// TIA Portal project "PLCII_Pro7" (V15.1)

(* hardware
DEVICE "S7-1200 station_1"  S7-1200 Station
   slot 0: "Rack_0"  S7-1200 Rack  Rack  V1.0
   slot 1: "PLC_1"  CPU 1215C DC/DC/Rly  6ES7 215-1HG40-0XB0  V4.2
*)

// ===== PLC "PLC_1"  CPU 1215C DC/DC/Rly =====

VAR_GLOBAL   // PLC tag table "Default tag table"
   "Start" AT %M0.0 : Bool;
   "Sys_runing" AT %M0.1 : Bool;
   "Stop" AT %M0.2 : Bool;
   "Activate" AT %M0.3 : Bool;
   "Sys_Activated" AT %M0.4 : Bool;
END_VAR

DATA_BLOCK "SysVaribales"   // DB1
{ S7_Optimized_Access := 'TRUE' }
VERSION : 0.1
   VAR
      StartSampling : Bool;
      StopSampling : Bool;
      SamplingRuning : Bool;
      StartCalibraton : Bool;
      StopCalibration : Bool;
      CalibrationRuning : Bool;
      O2Concentration : Int;
      O2ConcentrationMesuered : Int;
      O2_30Valve : Bool;
      O2_00Valve : Bool;
      StartCalibrationSeq : Bool;
      CalibrationDone : Bool;
      ScaleInputMIN : Int;
      ScaleInputMAX : Int := 0;
      O2_Zero_Average : Int;
      "O2_Maximum_ Concentration" : Int;
      "O2_Calibration_Gas_ Concentration" : Int;
      O2_Test_Gas_Average : Int;
      O2_Mesured : Int;
      O2_Concentration : Int;
   END_VAR
BEGIN
END_DATA_BLOCK

DATA_BLOCK "Sampling&&Calibration_DB"   // DB2
{ S7_Optimized_Access := 'TRUE' }
VERSION : 0.1
// stored: InstanceOfName Sampling&&Calibration
"Sampling&&Calibration"
BEGIN
END_DATA_BLOCK

DATA_BLOCK "ActuateValves_DB"   // DB5
{ S7_Optimized_Access := 'TRUE' }
VERSION : 0.1
// stored: InstanceOfName Calibration
"Calibration"
BEGIN
END_DATA_BLOCK

DATA_BLOCK "Calibration_DB"   // DB6
{ S7_Optimized_Access := 'TRUE' }
VERSION : 0.1
// stored: InstanceOfName Calibration
"Calibration"
BEGIN
END_DATA_BLOCK

DATA_BLOCK "Sampling_DB"   // DB7
{ S7_Optimized_Access := 'TRUE' }
VERSION : 0.1
// stored: InstanceOfName Sampling
"Sampling"
BEGIN
END_DATA_BLOCK

// folder: System blocks/Program resources

DATA_BLOCK "IEC_Timer_0_DB"   // DB3
{ S7_Optimized_Access := 'TRUE' }
AUTHOR : Simatic
FAMILY : IEC
NAME : IEC_TMR
VERSION : 1.0
// stored: InstanceOfName IEC_TIMER
"IEC_TIMER"
BEGIN
END_DATA_BLOCK

DATA_BLOCK "IEC_Timer_0_DB_1"   // DB4
{ S7_Optimized_Access := 'TRUE' }
AUTHOR : Simatic
FAMILY : IEC
NAME : IEC_TMR
VERSION : 1.0
// stored: InstanceOfName IEC_TIMER
"IEC_TIMER"
BEGIN
END_DATA_BLOCK

// folder: (top level)

FUNCTION_BLOCK "Sampling&&Calibration"   // FB1, LAD
{ S7_Optimized_Access := 'TRUE' }
VERSION : 0.1
   VAR_INPUT
      O2_Measured : Int;
   END_VAR
   VAR_OUTPUT
      O2_Concenetration : Real;
   END_VAR
   VAR
      ons1 : Bool;
      ons2 : Bool;
      ons3 : Bool;
      ons4 : Bool;
      ons5 : Bool;
      ons6 : Bool;
      ons7 : Bool;
      ons8 : Bool;
      ons9 : Bool;
      ons10 : Bool;
      ons11 : Bool;
   END_VAR
   VAR_TEMP
      O2_ValueTreated : Real;
   END_VAR
   VAR_TEMP   // added for the SCL form of the ladder/FBD networks
      _w1 : Bool;
   END_VAR
BEGIN

REGION Network 1
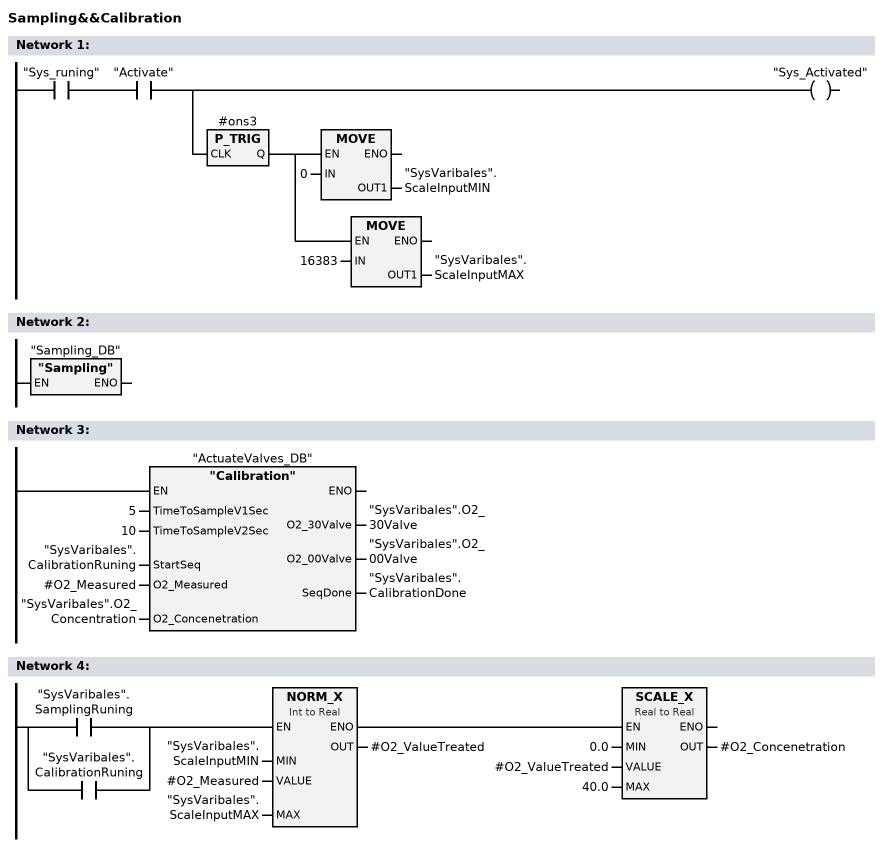
   RUNG wire#powerrail
      Contact( "Sys_runing" )
      Contact( "Activate" )
      wire#w1
      Coil( "Sys_Activated" )
   END_RUNG
   RUNG wire#w1
      P_Trig( #ons3 )
      wire#w2
      Move(in := 0, out1 => "SysVaribales".ScaleInputMIN)
   END_RUNG
   RUNG wire#w2
      Move(in := 16383, out1 => "SysVaribales".ScaleInputMAX)
   END_RUNG
   // the same network as SCL:
   "Sys_Activated" := "Sys_runing" AND "Activate";
   #_w1 := "Sys_Activated" AND NOT #ons3;   // rising edge
   #ons3 := "Sys_Activated";
   IF #_w1 THEN
       "SysVaribales".ScaleInputMIN := 0;
       "SysVaribales".ScaleInputMAX := 16383;
   END_IF;
END_REGION

REGION Network 2
   RUNG wire#powerrail
      "Sampling_DB"()
   END_RUNG
   // the same network as SCL:
   "Sampling_DB"();   // "Sampling"
END_REGION

REGION Network 3
   RUNG wire#powerrail
      "ActuateValves_DB"(TimeToSampleV1Sec := 5, TimeToSampleV2Sec := 10, StartSeq := "SysVaribales".CalibrationRuning, O2_Measured := #O2_Measured, O2_Concenetration := "SysVaribales".O2_Concentration, O2_30Valve => "SysVaribales".O2_30Valve, O2_00Valve => "SysVaribales".O2_00Valve, SeqDone => "SysVaribales".CalibrationDone)
   END_RUNG
   // the same network as SCL:
   "ActuateValves_DB"(TimeToSampleV1Sec := 5,   // "Calibration"
                      TimeToSampleV2Sec := 10,
                      StartSeq := "SysVaribales".CalibrationRuning,
                      O2_Measured := #O2_Measured,
                      O2_Concenetration := "SysVaribales".O2_Concentration,
                      O2_30Valve => "SysVaribales".O2_30Valve,
                      O2_00Valve => "SysVaribales".O2_00Valve,
                      SeqDone => "SysVaribales".CalibrationDone);
END_REGION

REGION Network 4
   RUNG wire#powerrail
      Contact( "SysVaribales".SamplingRuning )
      wire#w1
      { S7_Templates := "[SrcType := Int, DestType := Real]" } Normalize(min := "SysVaribales".ScaleInputMIN, value := #O2_Measured, max := "SysVaribales".ScaleInputMAX, out => #O2_ValueTreated)
      { S7_Templates := "[SrcType := Real, DestType := Real]" } Scale(min := 0.0, value := #O2_ValueTreated, max := 40.0, out => #O2_Concenetration)
   END_RUNG
   RUNG wire#powerrail
      Contact( "SysVaribales".CalibrationRuning )
   END_RUNG wire#w1
   // the same network as SCL:
   IF "SysVaribales".SamplingRuning OR "SysVaribales".CalibrationRuning THEN
       #O2_ValueTreated := NORM_X(MIN := "SysVaribales".ScaleInputMIN, VALUE := #O2_Measured, MAX := "SysVaribales".ScaleInputMAX);
       #O2_Concenetration := SCALE_X(MIN := 0.0, VALUE := #O2_ValueTreated, MAX := 40.0);
   END_IF;
END_REGION
END_FUNCTION_BLOCK

FUNCTION_BLOCK "Calibration"   // FB2, LAD
{ S7_Optimized_Access := 'TRUE' }
VERSION : 0.1
   VAR_INPUT
      TimeToSampleV1Sec : Int;
      TimeToSampleV2Sec : Int;
      StartSeq : Bool;
      O2_Measured : Int;
   END_VAR
   VAR_OUTPUT
      O2_30Valve : Bool;
      O2_00Valve : Bool;
      SeqDone : Bool;
   END_VAR
   VAR_IN_OUT
      O2_Concenetration : Int;
   END_VAR
   VAR
      startSecValve : Bool;
      ons1 : Bool;
      ons2 : Bool;
      ons3 : Bool;
      ons4 : Bool;
      ons5 : Bool;
      ons6 : Bool;
      ons7 : Bool;
      ons8 : Bool;
      UsedTIme1 : Time;
      UsedTIme2 : Time;
      O2_ValueTreated2 : Real;
   END_VAR
   VAR_TEMP
      TimeTemp1 : Int;
      UsedTimeTemp1 : Time;
      TimeTemp2 : Int;
      UsedTimeTemp2 : Time;
      O2_ValueTreated : Real;
      O2_30Average_MaxScaleTemp : Int;
      "O2_Maximum_ ConcentrationTemp" : Int;
      ScaleInputMAXTemp : Int;
      ScaleInputMAXTempReal : Real;
      ScaleInputMAXTempINT : Int;
   END_VAR
   VAR_TEMP   // added for the SCL form of the ladder/FBD networks
      _w1 : Bool;
      _w2 : Bool;
   END_VAR
BEGIN

REGION Network 1
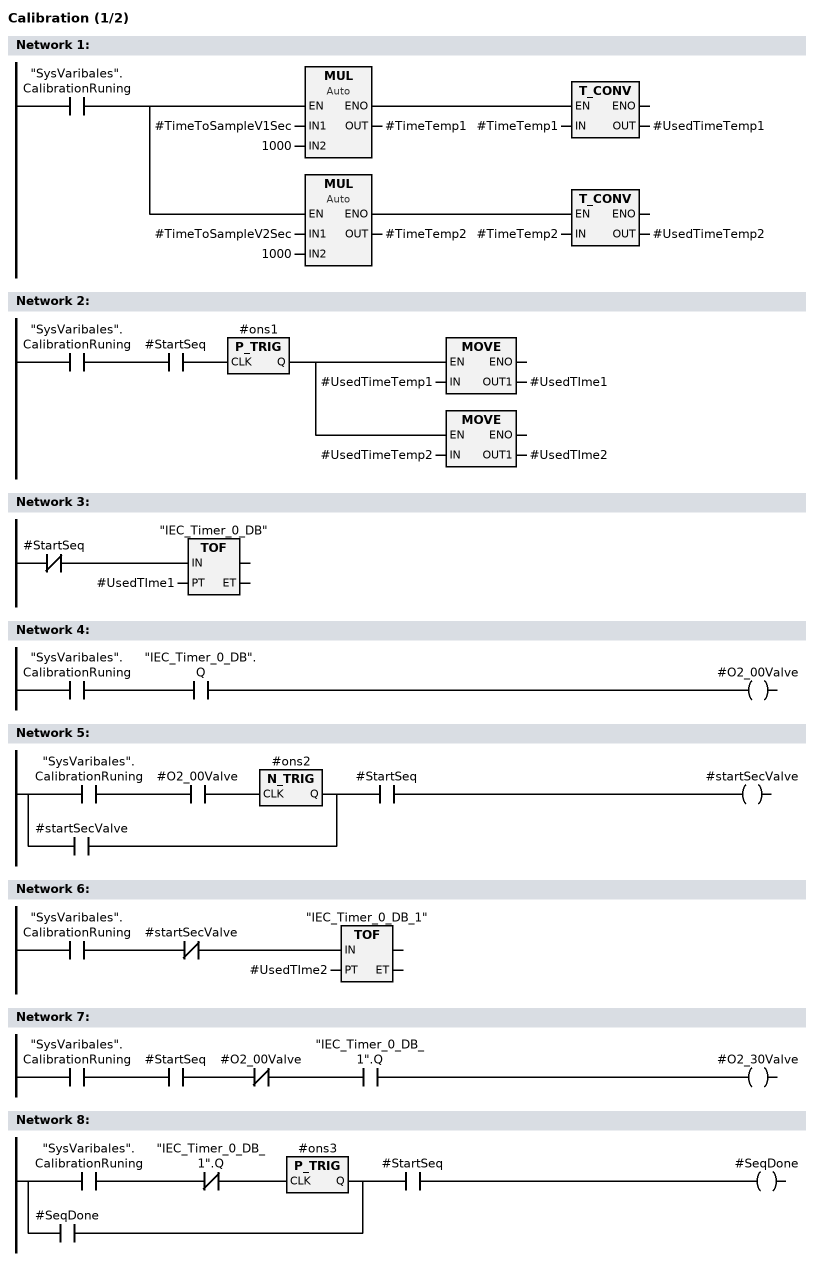
   IF "SysVaribales".CalibrationRuning THEN #TimeTemp1 := #TimeToSampleV1Sec * 1000; END_IF;
   #_w1 := "SysVaribales".CalibrationRuning;
   IF #_w1 THEN
       #UsedTimeTemp1 := T_CONV(IN := #TimeTemp1);
       #TimeTemp2 := #TimeToSampleV2Sec * 1000;
       #UsedTimeTemp2 := T_CONV(IN := #TimeTemp2);
   END_IF;
END_REGION

REGION Network 2
   RUNG wire#powerrail
      Contact( "SysVaribales".CalibrationRuning )
      Contact( #StartSeq )
      P_Trig( #ons1 )
      wire#w1
      Move(in := #UsedTimeTemp1, out1 => #UsedTIme1)
   END_RUNG
   RUNG wire#w1
      Move(in := #UsedTimeTemp2, out1 => #UsedTIme2)
   END_RUNG
   // the same network as SCL:
   #_w1 := "SysVaribales".CalibrationRuning AND #StartSeq;
   #_w2 := #_w1 AND NOT #ons1;   // rising edge
   #ons1 := #_w1;
   IF #_w2 THEN
       #UsedTIme1 := #UsedTimeTemp1;
       #UsedTIme2 := #UsedTimeTemp2;
   END_IF;
END_REGION

REGION Network 3
   "IEC_Timer_0_DB".TOF(IN := NOT #StartSeq, PT := #UsedTIme1);
END_REGION

REGION Network 4
   RUNG wire#powerrail
      Contact( "SysVaribales".CalibrationRuning )
      Contact( "IEC_Timer_0_DB".Q )
      Coil( #O2_00Valve )
   END_RUNG
   // the same network as SCL:
   #O2_00Valve := "SysVaribales".CalibrationRuning AND "IEC_Timer_0_DB".Q;
END_REGION

REGION Network 5
   RUNG wire#powerrail
      Contact( "SysVaribales".CalibrationRuning )
      Contact( #O2_00Valve )
      N_Trig( #ons2 )
      wire#w1
      Contact( #StartSeq )
      Coil( #startSecValve )
   END_RUNG
   RUNG wire#powerrail
      Contact( #startSecValve )
   END_RUNG wire#w1
   // the same network as SCL:
   #_w1 := "SysVaribales".CalibrationRuning AND #O2_00Valve;
   #_w2 := NOT #_w1 AND #ons2;   // falling edge
   #ons2 := #_w1;
   #startSecValve := (#_w2 OR #startSecValve) AND #StartSeq;
END_REGION

REGION Network 6
   "IEC_Timer_0_DB_1".TOF(IN := "SysVaribales".CalibrationRuning AND NOT #startSecValve, PT := #UsedTIme2);
END_REGION

REGION Network 7
   RUNG wire#powerrail
      Contact( "SysVaribales".CalibrationRuning )
      Contact( #StartSeq )
      I_Contact( #O2_00Valve )
      Contact( "IEC_Timer_0_DB_1".Q )
      Coil( #O2_30Valve )
   END_RUNG
   // the same network as SCL:
   #O2_30Valve := "SysVaribales".CalibrationRuning AND #StartSeq AND NOT #O2_00Valve AND "IEC_Timer_0_DB_1".Q;
END_REGION

REGION Network 8
   RUNG wire#powerrail
      Contact( "SysVaribales".CalibrationRuning )
      I_Contact( "IEC_Timer_0_DB_1".Q )
      P_Trig( #ons3 )
      wire#w1
      Contact( #StartSeq )
      Coil( #SeqDone )
   END_RUNG
   RUNG wire#powerrail
      Contact( #SeqDone )
   END_RUNG wire#w1
   // the same network as SCL:
   #_w1 := "SysVaribales".CalibrationRuning AND NOT "IEC_Timer_0_DB_1".Q;
   #_w2 := #_w1 AND NOT #ons3;   // rising edge
   #ons3 := #_w1;
   #SeqDone := (#_w2 OR #SeqDone) AND #StartSeq;
END_REGION

REGION Network 9
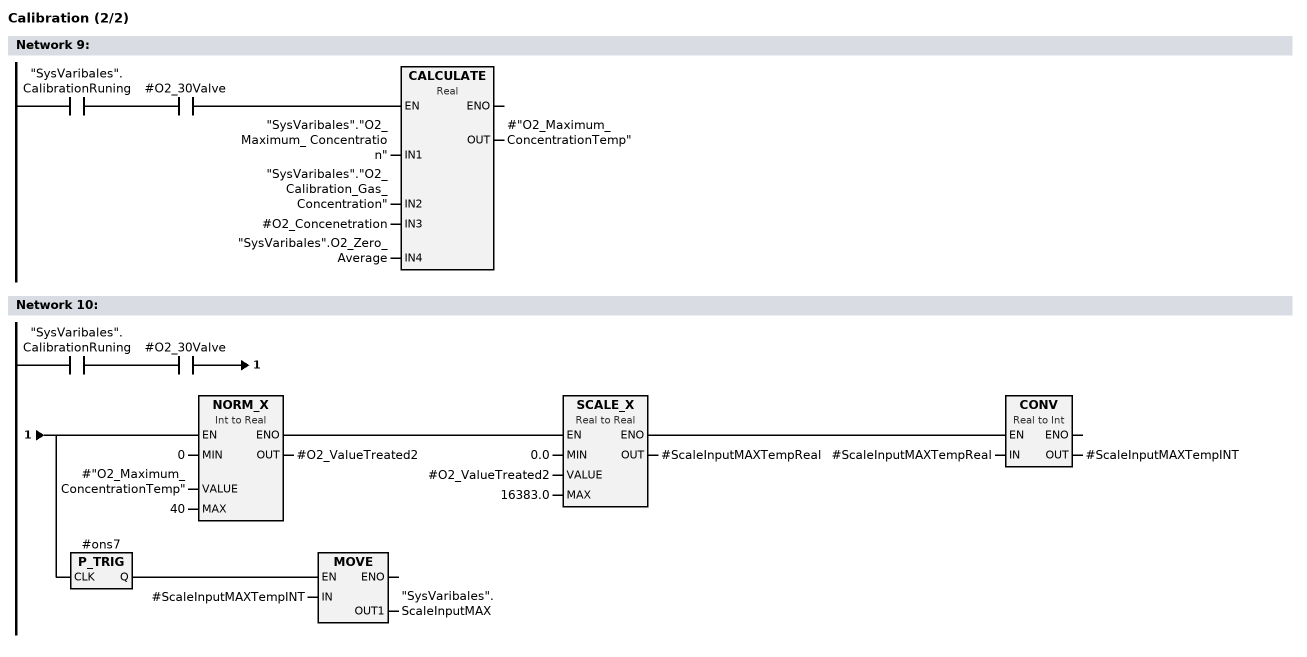
   RUNG wire#powerrail
      Contact( "SysVaribales".CalibrationRuning )
      Contact( #O2_30Valve )
      { S7_Templates := "SrcType := Real"; S7_Expression := "((IN1/IN2)*(IN3-IN4)) + IN4" } Calculate(in1 := "SysVaribales"."O2_Maximum_ Concentration", in2 := "SysVaribales"."O2_Calibration_Gas_ Concentration", in3 := #O2_Concenetration, in4 := "SysVaribales".O2_Zero_Average, out => #"O2_Maximum_ ConcentrationTemp")
   END_RUNG
   // the same network as SCL:
   IF "SysVaribales".CalibrationRuning AND #O2_30Valve THEN
       #"O2_Maximum_ ConcentrationTemp" := (("SysVaribales"."O2_Maximum_ Concentration"/"SysVaribales"."O2_Calibration_Gas_ Concentration")*(#O2_Concenetration-"SysVaribales".O2_Zero_Average)) + "SysVaribales".O2_Zero_Average;
   END_IF;
END_REGION

REGION Network 10
   RUNG wire#powerrail
      Contact( "SysVaribales".CalibrationRuning )
      Contact( #O2_30Valve )
      wire#w1
      { S7_Templates := "[SrcType := Int, DestType := Real]" } Normalize(min := 0, value := #"O2_Maximum_ ConcentrationTemp", max := 40, out => #O2_ValueTreated2)
      { S7_Templates := "[SrcType := Real, DestType := Real]" } Scale(min := 0.0, value := #O2_ValueTreated2, max := 16383.0, out => #ScaleInputMAXTempReal)
      { S7_Templates := "[SrcType := Real, DestType := Int]" } Convert(in := #ScaleInputMAXTempReal, out => #ScaleInputMAXTempINT)
   END_RUNG
   RUNG wire#w1
      P_Trig( #ons7 )
      Move(in := #ScaleInputMAXTempINT, out1 => "SysVaribales".ScaleInputMAX)
   END_RUNG
   // the same network as SCL:
   #_w1 := "SysVaribales".CalibrationRuning AND #O2_30Valve;
   IF #_w1 THEN
       #O2_ValueTreated2 := NORM_X(MIN := 0, VALUE := #"O2_Maximum_ ConcentrationTemp", MAX := 40);
       #ScaleInputMAXTempReal := SCALE_X(MIN := 0.0, VALUE := #O2_ValueTreated2, MAX := 16383.0);
       #ScaleInputMAXTempINT := REAL_TO_INT(#ScaleInputMAXTempReal);
   END_IF;
   #_w2 := #_w1 AND NOT #ons7;   // rising edge
   #ons7 := #_w1;
   IF #_w2 THEN "SysVaribales".ScaleInputMAX := #ScaleInputMAXTempINT; END_IF;
END_REGION
END_FUNCTION_BLOCK

FUNCTION_BLOCK "Sampling"   // FB3, LAD
{ S7_Optimized_Access := 'TRUE' }
VERSION : 0.1
   VAR
      ons1 : Bool;
      ons2 : Bool;
      ons3 : Bool;
      ons4 : Bool;
      ons5 : Bool;
      ons6 : Bool;
      ons7 : Bool;
      ons8 : Bool;
   END_VAR
   VAR_TEMP   // added for the SCL form of the ladder/FBD networks
      _w1 : Bool;
   END_VAR
BEGIN

REGION Network 1
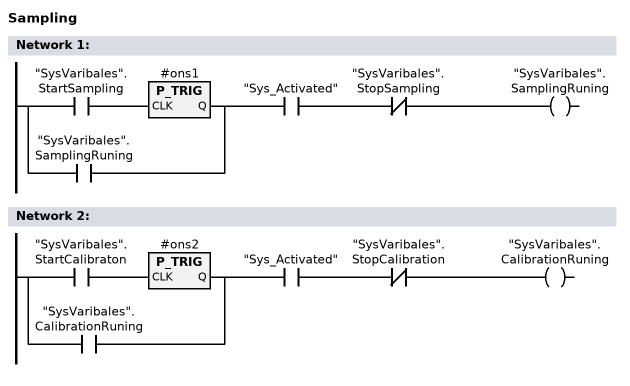
   RUNG wire#powerrail
      Contact( "SysVaribales".StartSampling )
      P_Trig( #ons1 )
      wire#w1
      Contact( "Sys_Activated" )
      I_Contact( "SysVaribales".StopSampling )
      Coil( "SysVaribales".SamplingRuning )
   END_RUNG
   RUNG wire#powerrail
      Contact( "SysVaribales".SamplingRuning )
   END_RUNG wire#w1
   // the same network as SCL:
   #_w1 := "SysVaribales".StartSampling AND NOT #ons1;   // rising edge
   #ons1 := "SysVaribales".StartSampling;
   "SysVaribales".SamplingRuning := (#_w1 OR "SysVaribales".SamplingRuning) AND "Sys_Activated" AND NOT "SysVaribales".StopSampling;
END_REGION

REGION Network 2
   RUNG wire#powerrail
      Contact( "SysVaribales".StartCalibraton )
      P_Trig( #ons2 )
      wire#w1
      Contact( "Sys_Activated" )
      I_Contact( "SysVaribales".StopCalibration )
      Coil( "SysVaribales".CalibrationRuning )
   END_RUNG
   RUNG wire#powerrail
      Contact( "SysVaribales".CalibrationRuning )
   END_RUNG wire#w1
   // the same network as SCL:
   #_w1 := "SysVaribales".StartCalibraton AND NOT #ons2;   // rising edge
   #ons2 := "SysVaribales".StartCalibraton;
   "SysVaribales".CalibrationRuning := (#_w1 OR "SysVaribales".CalibrationRuning) AND "Sys_Activated" AND NOT "SysVaribales".StopCalibration;
END_REGION
END_FUNCTION_BLOCK

ORGANIZATION_BLOCK "Main"   // OB1, LAD, ProgramCycle
TITLE = "Main Program Sweep (Cycle)"
{ S7_Optimized_Access := 'TRUE' }
VERSION : 0.1
   VAR_INPUT
      Initial_Call : Bool;   // Initial call of this OB
      Remanence : Bool;   // =True, if remanent data are available
   END_VAR
BEGIN

REGION Network 1
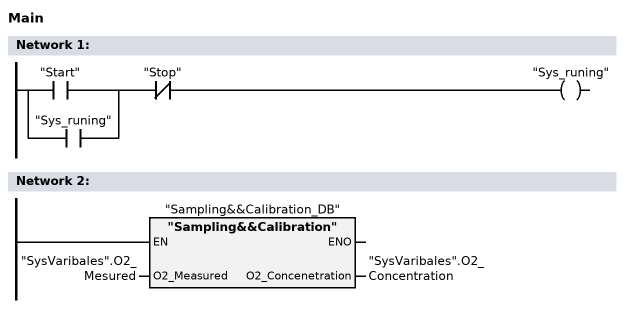
   RUNG wire#powerrail
      Contact( "Start" )
      wire#w1
      I_Contact( "Stop" )
      Coil( "Sys_runing" )
   END_RUNG
   RUNG wire#powerrail
      Contact( "Sys_runing" )
   END_RUNG wire#w1
   // the same network as SCL:
   "Sys_runing" := ("Start" OR "Sys_runing") AND NOT "Stop";
END_REGION

REGION Network 2
   RUNG wire#powerrail
      "Sampling&&Calibration_DB"(O2_Measured := "SysVaribales".O2_Mesured, O2_Concenetration => "SysVaribales".O2_Concentration)
   END_RUNG
   // the same network as SCL:
   "Sampling&&Calibration_DB"(O2_Measured := "SysVaribales".O2_Mesured,   // "Sampling&&Calibration"
                           O2_Concenetration => "SysVaribales".O2_Concentration);
END_REGION
END_ORGANIZATION_BLOCK